Universal Robots PolyScope program: Test Teach Position Peg.urp

Program Test Teach Position Peg (installation=default directory=/programs createdIn=5.21.3 lastSavedIn=5.21.3 robotSerialNumber=20246801938)
Calibrated DH parameters: a=[-0.000071, -0.790281, -0.600694, 0.000061, -0.000039, 0]; d=[0.236272, 604.465945, 132.116513, -736.382239, 0.159268, 0.154005]; alpha=[1.570254, -0.000567, 0.000559, 1.571709, -1.56999, 0]; deltaTheta=[0, -0.409357, 7.293326, -0.600784, -0.000001, -0.000001]
InitVariablesNode variables(variable(name=freedrive_m_var, expression=False))
Robot Program (runOnlyOnce=false)
  SuppressedNode
    MoveL speed 250 mm/s, acceleration 1200 mm/s^2 (useActiveTCP=true optimoveEnabled=false optiMoveSpeed=0.3 optiMoveAcceleration=0.09) feature=Base
      Waypoint Waypoint_1: TCP in base x=183.613 y=373.491 z=464.002 mm, rx=0 ry=3.1416 rz=0 rad; joints [-144.817, -120.486, 148.461, -117.931, -90.033, 125.101] deg; TCP offset x=0 y=0 z=19 mm, rx=0 ry=0 rz=0 rad
      'move welder up out of holder'
  MoveJ speed 60 deg/s, acceleration 80 deg/s^2 (useActiveTCP=false optimoveEnabled=false optiMoveSpeed=0.3 optiMoveAcceleration=0.09) tcp=TCP_1_plate; feature=Base
    Waypoint Waypoint_40: TCP in base x=360.688 y=270.12 z=646.145 mm, rx=0.0578 ry=2.126 rz=2.1341 rad; joints [-198.126, -117.852, 133.303, -13.01, -11.422, -6.036] deg
    'above waypoint is home'
    Waypoint Waypoint_2: TCP in base x=-548.957 y=386.285 z=143.71 mm, rx=1.5708 ry=0 rz=0 rad; joints [-60.253, -57.926, 123.544, -65.529, -60.311, -0.099] deg
  freedrive_m_var := False
  freedrive_m_var := True
  Popup Message (haltProgram=false message=Move the TCP to the top of the weld, then click 'Continue' inputType=Text)
  tcp_pose_top := get_actual_tcp_pose()
  Popup Message (haltProgram=false message=Move the TCP to the corner of the tank, then click 'Continue' inputType=Text)
  tcp_pose := get_actual_tcp_pose()
  freedrive_m_var := False
  Wait Sleep waitTime=0.25
  Script: sync()
